// TIA Portal V19 export
FUNCTION "RollfomrerLubr_CALL" : Void   // FC186, LAD
// stored: SetENOAutomatically false
BEGIN

REGION Network 1: Manager
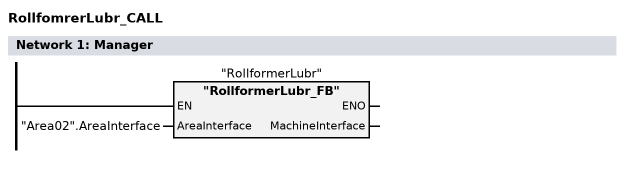
   RUNG wire#powerrail
      "RollformerLubr"(AreaInterface := "Area02".AreaInterface, MachineInterface =>)
   END_RUNG
   // the same network as SCL:
   "RollformerLubr"(AreaInterface := "Area02".AreaInterface);   // "RollformerLubr_FB"
END_REGION
END_FUNCTION
